// Mitsubishi GX Works2 project: 0722하던거2번   PLC: Q02/Q02H

PROGRAM MAIN
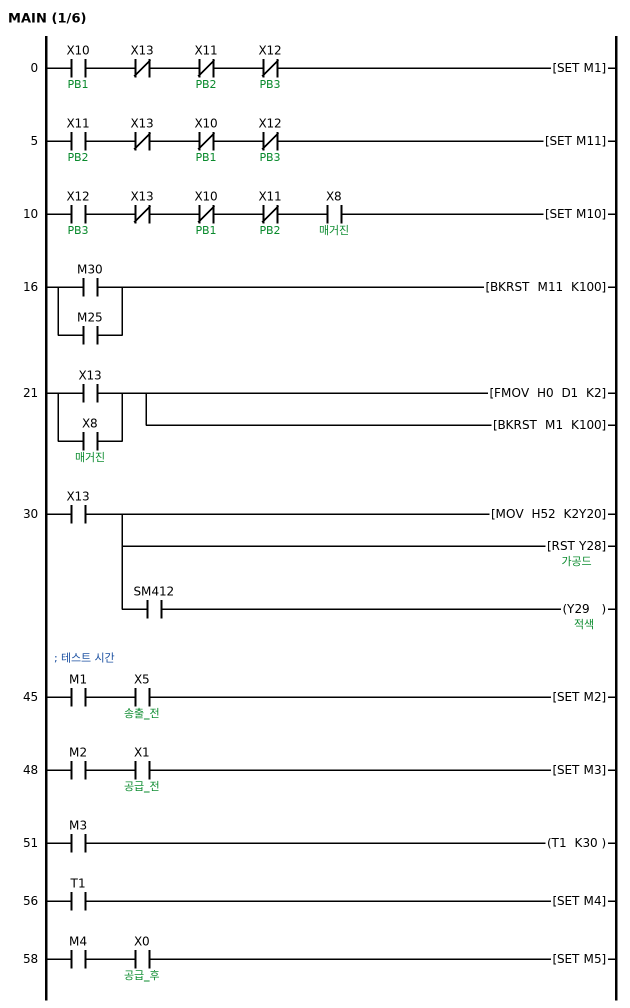
0     LD      X10  ; PB1
      ANI     X13
      ANI     X11  ; PB2
      ANI     X12  ; PB3
      SET     M1
5     LD      X11  ; PB2
      ANI     X13
      ANI     X10  ; PB1
      ANI     X12  ; PB3
      SET     M11
10    LD      X12  ; PB3
      ANI     X13
      ANI     X10  ; PB1
      ANI     X11  ; PB2
      AND     X8  ; 매거진
      SET     M10
16    LD      M30
      OR      M25
      BKRST   M11 K100
21    LD      X13
      OR      X8  ; 매거진
      FMOV    H0 D1 K2
      BKRST   M1 K100
30    LD      X13
      MOV     H52 K2Y20  ; 공급_전
      RST     Y28  ; 가공드
      AND     SM412
      OUT     Y29  ; 적색
; 테스트 시간
45    LD      M1
      AND     X5  ; 송출_전
      SET     M2
48    LD      M2
      AND     X1  ; 공급_전
      SET     M3
51    LD      M3
      OUT     T1 K30
56    LD      T1
      SET     M4
58    LD      M4
      AND     X0  ; 공급_후
      SET     M5
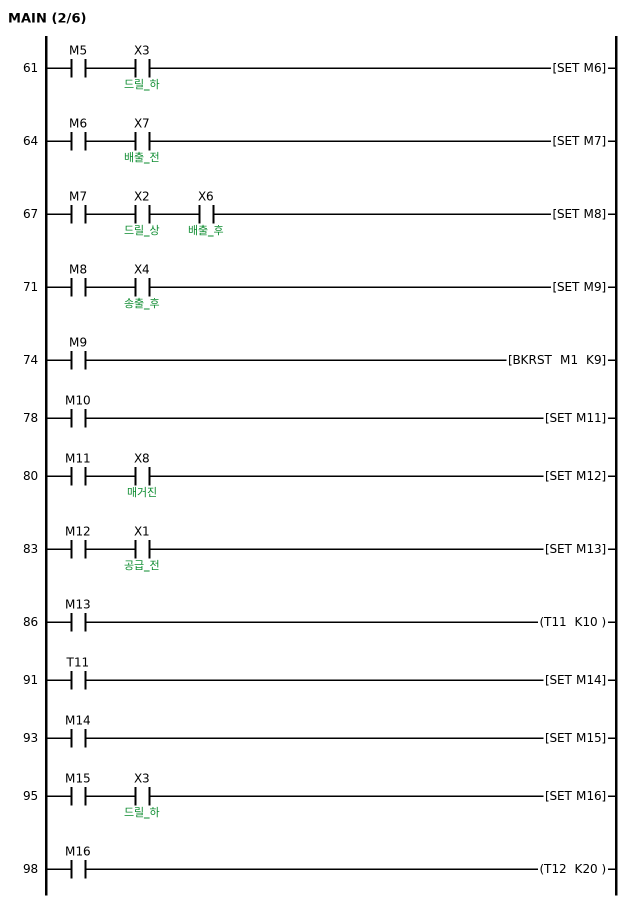
61    LD      M5
      AND     X3  ; 드릴_하
      SET     M6
64    LD      M6
      AND     X7  ; 배출_전
      SET     M7
67    LD      M7
      AND     X2  ; 드릴_상
      AND     X6  ; 배출_후
      SET     M8
71    LD      M8
      AND     X4  ; 송출_후
      SET     M9
74    LD      M9
      BKRST   M1 K9
78    LD      M10
      SET     M11
80    LD      M11
      AND     X8  ; 매거진
      SET     M12
83    LD      M12
      AND     X1  ; 공급_전
      SET     M13
86    LD      M13
      OUT     T11 K10
91    LD      T11
      SET     M14
93    LD      M14
      SET     M15
95    LD      M15
      AND     X3  ; 드릴_하
      SET     M16
98    LD      M16
      OUT     T12 K20
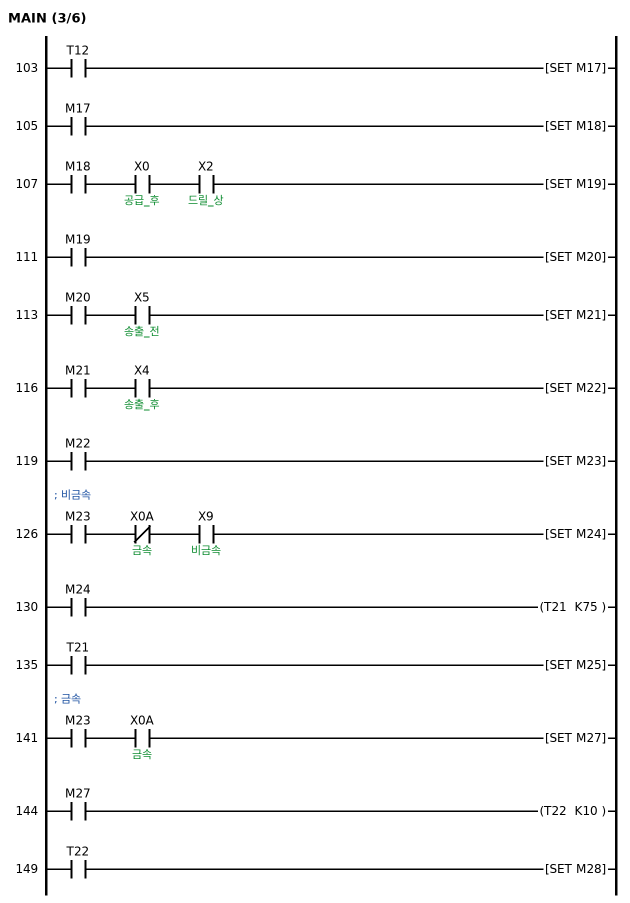
103   LD      T12
      SET     M17
105   LD      M17
      SET     M18
107   LD      M18
      AND     X0  ; 공급_후
      AND     X2  ; 드릴_상
      SET     M19
111   LD      M19
      SET     M20
113   LD      M20
      AND     X5  ; 송출_전
      SET     M21
116   LD      M21
      AND     X4  ; 송출_후
      SET     M22
119   LD      M22
      SET     M23
; 비금속
126   LD      M23
      ANI     X0A  ; 금속
      AND     X9  ; 비금속
      SET     M24
130   LD      M24
      OUT     T21 K75
135   LD      T21
      SET     M25
; 금속
141   LD      M23
      AND     X0A  ; 금속
      SET     M27
144   LD      M27
      OUT     T22 K10
149   LD      T22
      SET     M28
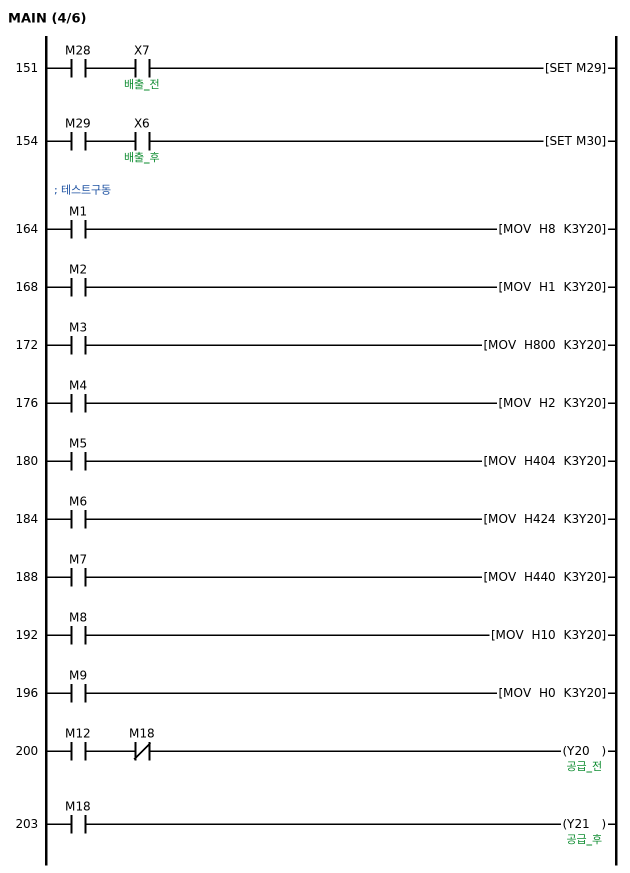
151   LD      M28
      AND     X7  ; 배출_전
      SET     M29
154   LD      M29
      AND     X6  ; 배출_후
      SET     M30
; 테스트구동
164   LD      M1
      MOV     H8 K3Y20
168   LD      M2
      MOV     H1 K3Y20
172   LD      M3
      MOV     H800 K3Y20
176   LD      M4
      MOV     H2 K3Y20
180   LD      M5
      MOV     H404 K3Y20
184   LD      M6
      MOV     H424 K3Y20
188   LD      M7
      MOV     H440 K3Y20
192   LD      M8
      MOV     H10 K3Y20
196   LD      M9
      MOV     H0 K3Y20
200   LD      M12
      ANI     M18
      OUT     Y20  ; 공급_전
203   LD      M18
      OUT     Y21  ; 공급_후
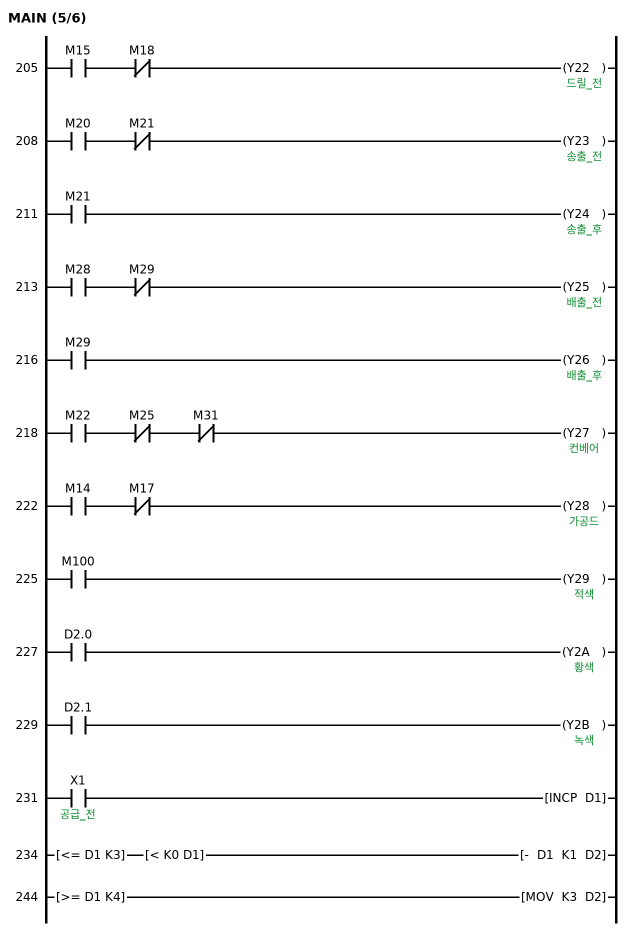
205   LD      M15
      ANI     M18
      OUT     Y22  ; 드릴_전
208   LD      M20
      ANI     M21
      OUT     Y23  ; 송출_전
211   LD      M21
      OUT     Y24  ; 송출_후
213   LD      M28
      ANI     M29
      OUT     Y25  ; 배출_전
216   LD      M29
      OUT     Y26  ; 배출_후
218   LD      M22
      ANI     M25
      ANI     M31
      OUT     Y27  ; 컨베어
222   LD      M14
      ANI     M17
      OUT     Y28  ; 가공드
225   LD      M100
      OUT     Y29  ; 적색
227   LD      D2.0
      OUT     Y2A  ; 황색
229   LD      D2.1
      OUT     Y2B  ; 녹색
231   LD      X1  ; 공급_전
      INCP    D1
234   LD<=    D1 K3
      AND<    K0 D1
      -       D1 K1 D2
244   LD>=    D1 K4
      MOV     K3 D2
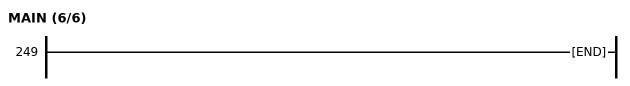
249   END
END_PROGRAM
